{attribute 'qualified_only'}
{attribute 'strict'}
TYPE XTSSequence :
(
	Off,
	EnableMovers,
	EnableGroup,
	AddAxes,
	RemoveAxes,
	RemovedAxes,
	DisableMovers,
	Disabled,
	Start,
	Run,
	Stop,
	Stopping,
	Pause,
	Pausing,
	Standby,
	Error,
	Waiting
);
END_TYPE

(* stored: Version 1.1.0.1, ProductVersion 3.1.4026.8
   EnumerationTextList XTSSequence: Id {46e9b238-637a-00fe-2d2b-4dec3a84e530} *)
